# EPICS autosave request: dxp/tags/R1-2/iocBoot/iocDxpLinux/auto_settings.req
file "mca_settings.req",                P=dxpLinux:, M=dxp_mca1
file "dxp_settings.req",                P=dxpLinux:, R=dxp1
